// TIA Portal project "Oransal_Kontrol_Uygulaması_V1" (V16)

(* hardware
DEVICE "S7-1200 station_1"  S7-1200 Station
   slot 0: "Rack_0"  S7-1200 Rack  Rack  V1.0
   slot 1: "PLC_1"  CPU 1214C DC/DC/DC  6ES7 214-1AG40-0XB0  V4.3
   slot 2: "AI 4xRTD_1"  SM 1231 AI4 x RTD  6ES7 231-5PD32-0XB0  V2.0
   slot 3: "AQ 4x14BIT_1"  6ES7 232-4HD32-0XB0  V2.1
*)

// ===== PLC "PLC_1"  CPU 1214C DC/DC/DC =====

VAR_GLOBAL   // PLC tag table "Default tag table"
   "Set_Değeri" AT %MW10 : Int;
   "PT100" AT %IW96 : Int;
   "Kat_Sayı" AT %MD12 : Real;
   "Üst" AT %MD16 : Real;
   "Alt" AT %MD20 : Real;
   "Oransal_Kontrol_Çıkışı" AT %MD24 : Real;
   "NormX_Çıkışı" AT %MD28 : Real;
   "Sıcaklık_Çıkışı" AT %QW112 : Int;
END_VAR

DATA_BLOCK "Oransal Kontrol_DB"   // DB1
{ S7_Optimized_Access := 'TRUE' }
VERSION : 0.1
// stored: InstanceOfName Oransal Kontrol
"Oransal Kontrol"
BEGIN
END_DATA_BLOCK

FUNCTION_BLOCK "Oransal Kontrol"   // FB1, LAD
{ S7_Optimized_Access := 'TRUE' }
VERSION : 0.1
   VAR_INPUT
      Set_Değeri : Int;
      gerçek_Değer : Int;
      Oransal_Katsayı : Real;
      Üst_Limit_1 : Real;
      Alt_Limit_1 : Real;
   END_VAR
   VAR_OUTPUT
      Çıkış : Real;
   END_VAR
   VAR
      Set_Değeri_Real : Real;
      Gerçek_Değeri_Real : Real;
      Gerçek_Sıcaklık_Real : Real;
      Sonuç_1 : Real;
      Sonuç_2 : Real;
   END_VAR
BEGIN

REGION Network 1: Set Değerini Real'a Çevirme
   // - Burada istediğimiz sıcaklık #Set_Değeri değişkeninde tutuluyor
   //    .
   // 
   // #Set_Değeri = 50 
   // 
   // 
   //     Ancak bu değişkenin veri tipi INT, yani tam sayıdır. İleride ondalıklı hesap yapabilmek için CONV         komutuyla REAL veri tipine çevrilir:
   // 
   // 
   //     50 → 50.0
   // 
   // 
   //     Sonuç:
   // 
   // 
   //     #Set_Değeri_Real = 50.0
   // 
   // 
   //     Bu Network sıcaklığı değiştirmez. Yalnızca sayının veri tipini değiştirir.
   //     
   // 
   // Network 1’in görevi: İstenen sıcaklığı hesaplamalarda kullanılabilmesi için INT’den REAL’e         çevirmek.
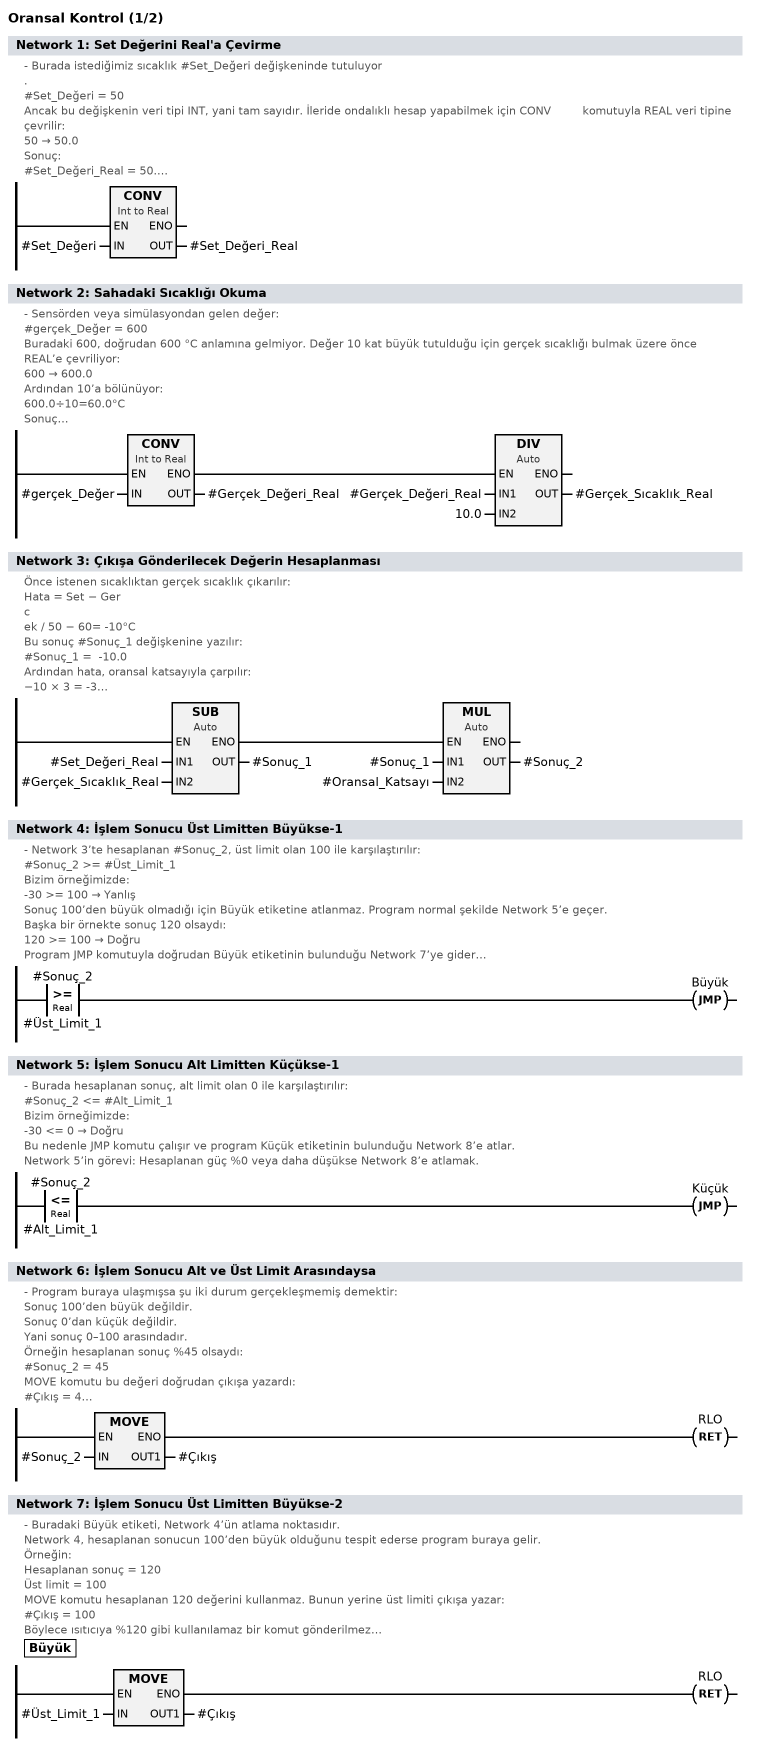
   RUNG wire#powerrail
      { S7_Templates := "[SrcType := Int, DestType := Real]" } Convert(in := #Set_Değeri, out => #Set_Değeri_Real)
   END_RUNG
   // the same network as SCL:
   #Set_Değeri_Real := INT_TO_REAL(#Set_Değeri);
END_REGION

REGION Network 2: Sahadaki Sıcaklığı Okuma
   // - Sensörden veya simülasyondan gelen değer:
   //     
   // 
   // #gerçek_Değer = 600
   // 
   // 
   //     Buradaki 600, doğrudan 600 °C anlamına gelmiyor. Değer 10 kat büyük tutulduğu için gerçek sıcaklığı bulmak üzere önce REAL’e çevriliyor:
   //     
   // 
   // 600 → 600.0
   // 
   // 
   //     Ardından 10’a bölünüyor:
   // 
   // 
   //     600.0÷10=60.0°C
   // 
   // 
   //     Sonuç:
   //     #Gerçek_Sıcaklık_Real = 60.0
   // 
   // 
   //     Network 2’nin görevi: Sensörden gelen 600 değerini 60 °C olarak kullanılabilecek hâle getirmek.
   RUNG wire#powerrail
      { S7_Templates := "[SrcType := Int, DestType := Real]" } Convert(in := #gerçek_Değer, out => #Gerçek_Değeri_Real)
      Div(in1 := #Gerçek_Değeri_Real, in2 := 10.0, out => #Gerçek_Sıcaklık_Real)
   END_RUNG
   // the same network as SCL:
   #Gerçek_Değeri_Real := INT_TO_REAL(#gerçek_Değer);
   #Gerçek_Sıcaklık_Real := #Gerçek_Değeri_Real / 10.0;
END_REGION

REGION Network 3: Çıkışa Gönderilecek Değerin Hesaplanması
   // Önce istenen sıcaklıktan gerçek sıcaklık çıkarılır:
   // 
   // Hata = Set − Ger
   // c
   // ek / 50 − 60= -10°C
   // 
   // 
   // Bu sonuç #Sonuç_1 değişkenine yazılır:
   // 
   // 
   // #Sonuç_1 =  -10.0
   // 
   // 
   // Ardından hata, oransal katsayıyla çarpılır:
   // 
   // 
   // −10 × 3 = -30
   // 
   // 
   // Sonuç:
   // 
   // 
   // #Sonuç_2 = -30.0
   // 
   // 
   // Bu, programın hesapladığı ilk kontrol çıkışıdır. Ancak henüz çıkışa gönderilemez; çünkü belirlediğimiz 0–100 sınırlarının dışındadır.
   // 
   // 
   // Network 3’ün görevi: Sıcaklık hatasını bulmak ve hatayı oransal katsayıyla çarparak gerekli ısıtıcı gücünü hesaplamak.
   // 
   // Temel formül:
   // 
   //  (cıkıs= (Set - Gercek) x Kp​
   RUNG wire#powerrail
      Sub(in1 := #Set_Değeri_Real, in2 := #Gerçek_Sıcaklık_Real, out => #Sonuç_1)
      Mul(in1 := #Sonuç_1, in2 := #Oransal_Katsayı, out => #Sonuç_2)
   END_RUNG
   // the same network as SCL:
   #Sonuç_1 := #Set_Değeri_Real - #Gerçek_Sıcaklık_Real;
   #Sonuç_2 := #Sonuç_1 * #Oransal_Katsayı;
END_REGION

REGION Network 4: İşlem Sonucu Üst Limitten Büyükse-1
   // - Network 3’te hesaplanan #Sonuç_2, üst limit olan 100 ile karşılaştırılır:
   // 
   // 
   // #Sonuç_2 >= #Üst_Limit_1
   // 
   // 
   // Bizim örneğimizde:
   // 
   // 
   // -30 >= 100 → Yanlış
   // 
   // 
   // Sonuç 100’den büyük olmadığı için Büyük etiketine atlanmaz. Program normal şekilde Network 5’e geçer.
   // 
   // 
   // Başka bir örnekte sonuç 120 olsaydı:
   // 
   // 
   // 120 >= 100 → Doğru
   // 
   // 
   // Program JMP komutuyla doğrudan Büyük etiketinin bulunduğu Network 7’ye gider.
   // 
   // 
   // Network 4’ün görevi: Hesaplanan güç %100 veya daha fazlaysa Network 7’ye atlamak.
   RUNG wire#powerrail
      { S7_Templates := "SrcType := Real" } GE_Contact(in1 := #Sonuç_2, in2 := #Üst_Limit_1)
      JumpCoil( Büyük )
   END_RUNG
   // the same network as SCL:
   IF #Sonuç_2 >= #Üst_Limit_1 THEN GOTO Büyük; END_IF;
END_REGION

REGION Network 5: İşlem Sonucu Alt Limitten Küçükse-1
   // - Burada hesaplanan sonuç, alt limit olan 0 ile karşılaştırılır:
   // 
   // #Sonuç_2 <= #Alt_Limit_1
   // 
   // Bizim örneğimizde:
   // 
   // -30 <= 0 → Doğru
   // 
   // Bu nedenle JMP komutu çalışır ve program Küçük etiketinin bulunduğu Network 8’e atlar.
   // 
   // Network 5’in görevi: Hesaplanan güç %0 veya daha düşükse Network 8’e atlamak.
   RUNG wire#powerrail
      { S7_Templates := "SrcType := Real" } LE_Contact(in1 := #Sonuç_2, in2 := #Alt_Limit_1)
      JumpCoil( Küçük )
   END_RUNG
   // the same network as SCL:
   IF #Sonuç_2 <= #Alt_Limit_1 THEN GOTO Küçük; END_IF;
END_REGION

REGION Network 6: İşlem Sonucu Alt ve Üst Limit Arasındaysa
   // - Program buraya ulaşmışsa şu iki durum gerçekleşmemiş demektir:
   // 
   // Sonuç 100’den büyük değildir.
   // Sonuç 0’dan küçük değildir.
   // 
   // Yani sonuç 0–100 arasındadır.
   // 
   // Örneğin hesaplanan sonuç %45 olsaydı:
   // 
   // #Sonuç_2 = 45
   // 
   // MOVE komutu bu değeri doğrudan çıkışa yazardı:
   // 
   // #Çıkış = 45
   // 
   // Ardından RET komutu FB’nin çalışmasını sonlandırır. Böylece Network 7 ve Network 8 gereksiz yere çalıştırılmaz.
   // 
   // Bizim örneğimizde sonuç -30 olduğu için Network 5’ten Network 8’e atlandı; dolayısıyla Network 6 çalışmaz.
   // 
   // Network 6’nın görevi: Hesaplanan değer 0–100 arasındaysa değeri değiştirmeden çıkışa yazmak ve bloğu bitirmek.
   #Çıkış := #Sonuç_2;
   ENO := TRUE;
   RETURN;
END_REGION

REGION Network 7: İşlem Sonucu Üst Limitten Büyükse-2
   // - Buradaki Büyük etiketi, Network 4’ün atlama noktasıdır.
   // 
   // Network 4, hesaplanan sonucun 100’den büyük olduğunu tespit ederse program buraya gelir.
   // 
   // Örneğin:
   // 
   // Hesaplanan sonuç = 120
   // Üst limit = 100
   // 
   // MOVE komutu hesaplanan 120 değerini kullanmaz. Bunun yerine üst limiti çıkışa yazar:
   // 
   // #Çıkış = 100
   // 
   // Böylece ısıtıcıya %120 gibi kullanılamaz bir komut gönderilmez.
   // 
   // Ardından RET komutu bloğu bitirir.
   // 
   // Network 7’nin görevi: Hesaplanan güç %100’ü geçerse çıkışı en fazla %100 yapmak.
   Büyük:
   #Çıkış := #Üst_Limit_1;
   ENO := TRUE;
   RETURN;
END_REGION

REGION Network 8: İşlem Sonucu Alt Limitten Küçükse-2
   // - Buradaki Küçük etiketi, Network 5’in atlama noktasıdır.
   // 
   // Bizim örneğimizde hesaplanan sonuç:
   // 
   // #Sonuç_2 = -30
   // 
   // Alt limit:
   // 
   // #Alt_Limit_1 = 0
   // 
   // Network 5’te -30 <= 0 koşulu doğru olduğu için program Network 8’e atlar.
   // 
   // Buradaki MOVE komutu alt limiti çıkışa yazar:
   // 
   // #Çıkış = 0
   // 
   // Yani ısıtıcı kapatılır.
   // 
   // Network 8’in görevi: Hesaplanan güç sıfırın altına düşerse çıkışı %0 yapmak.
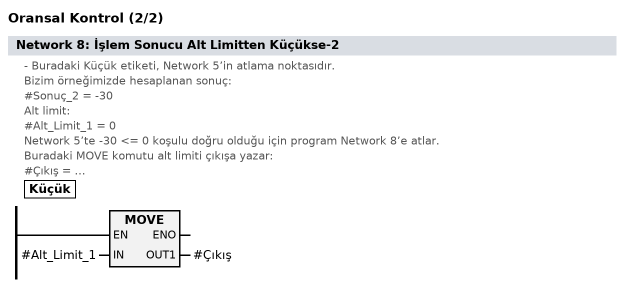
   Label( Küçük )
   RUNG wire#powerrail
      Move(in := #Alt_Limit_1, out1 => #Çıkış)
   END_RUNG
   // the same network as SCL:
   Küçük:
   #Çıkış := #Alt_Limit_1;
END_REGION
END_FUNCTION_BLOCK

ORGANIZATION_BLOCK "Main"   // OB1, LAD, ProgramCycle
TITLE = "Main Program Sweep (Cycle)"
{ S7_Optimized_Access := 'TRUE' }
VERSION : 0.1
   VAR_INPUT
      Initial_Call : Bool;   // Initial call of this OB
      Remanence : Bool;   // =True, if remanent data are available
   END_VAR
BEGIN

REGION Network 1: Oransal Kontrol Alt Programı
   // - Oransal kontrolde set noktasına yaklaşılmadan önce set noktası görülmeye çalışılır ve görülmeye başlandıktan sonra çıkış gücü yavaş yavaş kısılır. Nasıl ki kırmızı ışığı görmeye başladığımızda frene basıyoruz işte bu da böyle bir şey. Eğer kırmızı ışığın dibinde frene basarsanız bir yayaya çarparsınız. Oransal kontrolde de önceden set noktasını görmeden set noktasında gücü keserseniz set noktasından çok saparsınız.
   // 
   // Oransal kontrol de bir oransal bant oluşturuyoruz. Set değeri bu bandın ortası oluyor. Set değerinin öncesinde yani bandın başlangıç noktasında çıkış gücü kısılır. Set noktasına gelindiğinde çıkış gücü %50 olur. Bandın diğer ucuna gelindiğinde ise çıkış gücü artık sıfırdır.
   // 
   // İşte biz bu bandın genişliğini oransal katsayı ile belirliyoruz. Mesela set değerinin 100 olduğu bir sistemde, set değeri ile ölçülen değer arası 10 ise ve oransal katsayı da 3 ise bu durumda oransal bant 70 ten başlar ve 130 da biter. Siz bu oransal bandı oransal katsayı ile daraltıp genişletebilirsiniz. Bu bandı iyi ayarlamanız lazım yoksa set değerini tutturamazsınız.
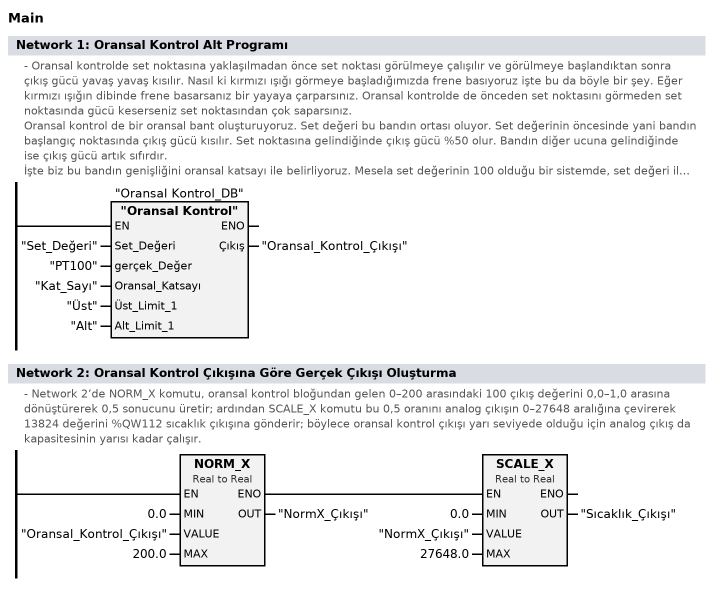
   RUNG wire#powerrail
      "Oransal Kontrol_DB"(Set_Değeri := "Set_Değeri", gerçek_Değer := "PT100", Oransal_Katsayı := "Kat_Sayı", Üst_Limit_1 := "Üst", Alt_Limit_1 := "Alt", Çıkış => "Oransal_Kontrol_Çıkışı")
   END_RUNG
   // the same network as SCL:
   "Oransal Kontrol_DB"(Set_Değeri := "Set_Değeri",   // "Oransal Kontrol"
                        gerçek_Değer := "PT100",
                        Oransal_Katsayı := "Kat_Sayı",
                        Üst_Limit_1 := "Üst",
                        Alt_Limit_1 := "Alt",
                        Çıkış => "Oransal_Kontrol_Çıkışı");
END_REGION

REGION Network 2: Oransal Kontrol Çıkışına Göre Gerçek Çıkışı Oluşturma
   // - Network 2’de NORM_X komutu, oransal kontrol bloğundan gelen 0–200 arasındaki 100 çıkış değerini 0,0–1,0 arasına dönüştürerek 0,5 sonucunu üretir; ardından SCALE_X komutu bu 0,5 oranını analog çıkışın 0–27648 aralığına çevirerek 13824 değerini %QW112 sıcaklık çıkışına gönderir; böylece oransal kontrol çıkışı yarı seviyede olduğu için analog çıkış da kapasitesinin yarısı kadar çalışır.
   RUNG wire#powerrail
      { S7_Templates := "[SrcType := Real, DestType := Real]" } Normalize(min := 0.0, value := "Oransal_Kontrol_Çıkışı", max := 200.0, out => "NormX_Çıkışı")
      { S7_Templates := "[SrcType := Real, DestType := Real]" } Scale(min := 0.0, value := "NormX_Çıkışı", max := 27648.0, out => "Sıcaklık_Çıkışı")
   END_RUNG
   // the same network as SCL:
   "NormX_Çıkışı" := NORM_X(MIN := 0.0, VALUE := "Oransal_Kontrol_Çıkışı", MAX := 200.0);
   "Sıcaklık_Çıkışı" := SCALE_X(MIN := 0.0, VALUE := "NormX_Çıkışı", MAX := 27648.0);
END_REGION
END_ORGANIZATION_BLOCK